(* CODESYS project Untitled1.project

Project tree, tasks and I/O mapping:
  Device : CODESYS Control Win V3, 3S - Smart Software Solutions GmbH, version 3.5.12.10
    application Application
      libraries: Standard, * (System)
      task MainTask (cyclic, interval t#20ms, priority 1) calls PLC_PRG
      task VISU_TASK (cyclic, interval 100 ms, priority 31) calls VisuElems.Visu_Prg
      program PLC_PRG [LD]
      visualisation Visualization
  text list GlobalTextList
*)

// Device/Application/PLC_PRG
PROGRAM PLC_PRG
VAR
	targetTemp: BOOL;
	START: BOOL;
	VALVE1: BOOL;
	FloatSwitch: BOOL;
	Heater: BOOL;
	VALVE2: BOOL;
	Timer: TON;
	elapsedTime: TIME;
	Alarm: BOOL;
END_VAR

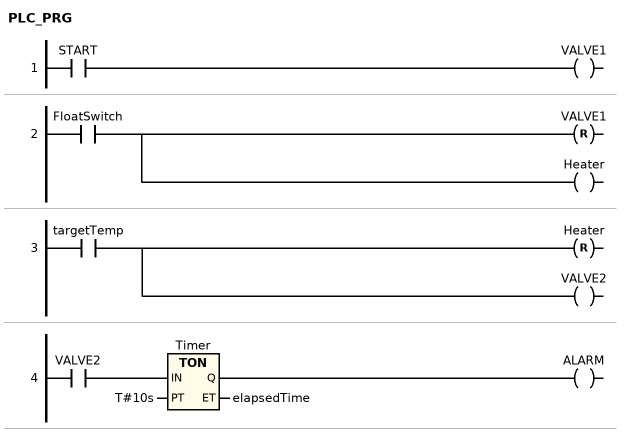
// NETWORK 1
VALVE1 := START;

// NETWORK 2
VALVE1 R= FloatSwitch;
Heater := FloatSwitch;

// NETWORK 3
Heater R= targetTemp;
VALVE2 := targetTemp;

// NETWORK 4
Timer(IN := VALVE2, PT := T#10s, ET => elapsedTime); // TON
ALARM := Timer.Q;

END_PROGRAM

// Device/Application/Visualization
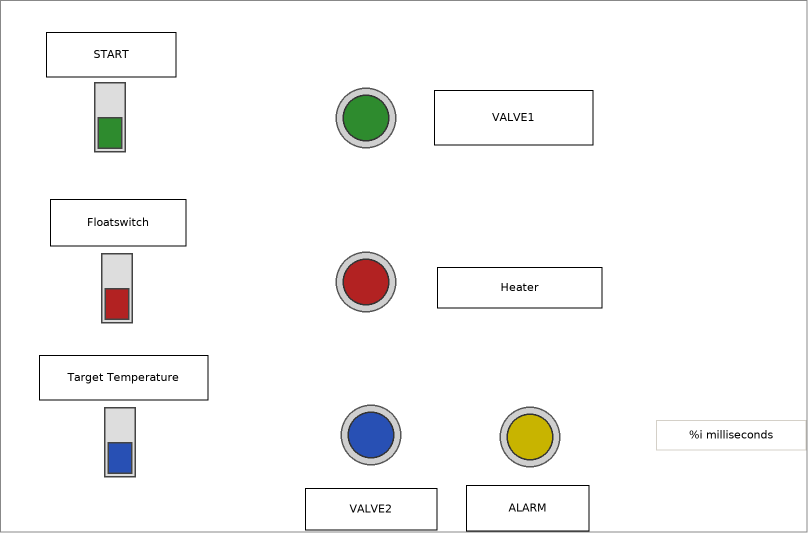
VISUALIZATION Visualization  // 808x533
    DipSwitch (75,82 70x70), variable: PLC_PRG.START, behaviour: TOGGLE, style: Switch-DipSwitch-Green
    Lamp1 (331,83 70x70), variable: PLC_PRG.VALVE1, style: Lamp-Lamp1-Green
    Rectangle (46,32 130x45), "START"
    Rectangle (434,90 159x55), "VALVE1"
    DipSwitch (82,253 70x70), variable: PLC_PRG.FloatSwitch, behaviour: TOGGLE, style: Switch-DipSwitch-Red
    Lamp1 (331,247 70x70), variable: PLC_PRG.Heater, style: Lamp-Lamp1-Red
    Rectangle (50,199 136x47), "Floatswitch"
    Rectangle (437,267 165x41), "Heater"
    Rectangle (305,488 132x42), "VALVE2"
    Rectangle (466,485 123x46), "ALARM"
    Lamp1 (495,402 70x70), variable: PLC_PRG.Alarm, style: Lamp-Lamp1-Yellow
    Lamp1 (336,400 70x70), variable: PLC_PRG.VALVE2, style: Lamp-Lamp1-Blue
    DipSwitch (85,407 70x70), variable: PLC_PRG.targetTemp, behaviour: TOGGLE, style: Switch-DipSwitch-Blue
    Rectangle (39,355 169x45), "Target Temperature"
    Textfield (656,420 150x30), "%i milliseconds", text variable: PLC_PRG.Timer.ET
END_VISUALIZATION
